// TIA Portal V19 export
TYPE "TAx_Speed_Sts"
// stored: Access Published
   STRUCT
      AlarmPresence : Bool;   // Cumulative alarm presence
      WarningPresence : Bool;   // Cumulative warning presence
      Enabled : Bool;   // Axis is enabled
      Done : Bool;
      Standstill : Bool;   // Axis is standstill
      RstHWDone : Bool;   // Reset hardware done
      AtProgrammedSpeed : Bool;
      MoveMinusPermitted : Bool;
      MovePlusPermitted : Bool;
      ActualSpeed : LReal;
   END_STRUCT;
END_TYPE
